(* Schneider Machine Expert - Basic project Shute_project, file version 2.2.0.0 *)
(* ProjectInformations: Name=Yeni proje *)

HARDWARE
  Cpu 0: TM221CE40R
  EthernetConfiguration: NetworkName=M221, IpAllocationMode=FixedAddress, IpAddress=0.0.0.0, SubnetMask=0.0.0.0
  SerialLineConfiguration: Baud=Baud19200, Parity=ParityEven, DataBits=DataBits8, StopBits=StopBits1, PhysicalMedium=PhysicalMediumRs485, TransmissionMode=TransmissionModeModbusRtu, SlaveId=1, Addressing=SlaveAddressing
  MastTask: UsePeriodScanMode=false, PeriodScan=100
  FastTask: Period=255
  CpuBehavior: StartingMode=StartAsPreviousState, AutoSaveRamOnEeprom=true, WatchdogPeriod=250

SYMBOLS  (address, symbol, comment, settings)
  %M0       K01_PERMISON
  %M1       K02_1_LOADING_ON
  %M2       K03_1_LEVEL_INDICATOR
  %M3       K04_1_TIMER
  %M4       K05_1_PARK_POSITION
  %M5       K06_1
  %M6       K07_1_SLACK_ROPE
  %M7       K08_1_LIFT_AUTO
  %M8       K11__1_LIFT_CHUTE
  %M9       K012_GAT1_O
  %M10      MAIN_CONTACTOR_1
  %M11      K017_1
  %M12      K12_1_OPEN_GATE
  %M13      K22_1_CLOSE_GATE
  %M14      K022_GATE_1_C
  %M15      LıFT_CHUTE_S63
  %M16      LOWER_CHUTE_S64
  %M17      LıFT_CHUTE_1
  %M18      LOADNG_ON
  %M19      K016_1_TIMER
  %M20      MAIN_CONTACTOR_2
  %M21      K07_2_SLACK_ROPE
  %M22      K02_2
  %M23      K06_2
  %M24      K05_2
  %M25      H62_LAMP
  %M26      ZS07_2
  %M27      K08_2
  %M28      K03_2
  %M29      K04_2
  %M30      LS01_2_SONDA_MAX_INPUT
  %M31      K012_2
  %M32      K022_2
  %M33      K016_2
  %M34      K017_2
  %I0.0     S61_EMERGENCY_OFF
  %I0.1     S62_EQUIPMENT_ON
  %I0.2     K100_K101_RELASE
  %I0.3     SLACK_ROPE_SENSOR_1
  %I0.4     LOADING_ON
  %I0.5     LOADING_OFF
  %I0.6     LIFT_CHUTE
  %I0.7     LOWER_CHUTE
  %I0.8     S65_LOADING_ON
  %I0.9     S66_LOADING_OFF
  %I0.10    ZS03_LIMIT_SWITCH_HOIST
  %I0.11    ZS07_LIMIT_PARK_SENSOR
  %I0.12    LS01_1_SONDA
  %I0.13    ZS01_1_LIMIT_SWITH_LOWER  "this should be 2zs01"
  %I0.14    GATE_1_1B11_O
  %I0.15    GATE_1_1B12
  %I0.16    GATE_2_2B11_O
  %I0.17    GATE_2_2B12_C
  %I0.18    S70_CHUTE_1
  %I0.19    S70_CHUTE_2
  %I0.20    ZS02_1
  %I0.21    SLACK_ROPE_SENSOR_2
  %I0.22    ZS02_2
  %I0.23    ZS072
  %Q0.0     H4_LAMP
  %Q0.1     H5_LAMP
  %Q0.2     H63_LAMP
  %Q0.3     K11_1_LIFT_CHUTE
  %Q0.4     K21_1_LOWER_CHUTE
  %Q0.5     K02_1_OUTPUT
  %Q0.6     K12_OPEN_GATE_1
  %Q0.7     K22_CLOSE_GATE_1
  %Q0.8     K11_2_LIFT_CHUTE
  %Q0.9     K12_2_LOWER_CHUTE
  %Q0.10    K02_2_OUTPUT
  %Q0.11    K12_OPEN_GATE_2
  %Q0.12    K22_2_CLOSE_GATE_2
  %Q0.13    K21_2

POU Yeni POU
  (* SectionNumber=1 *)

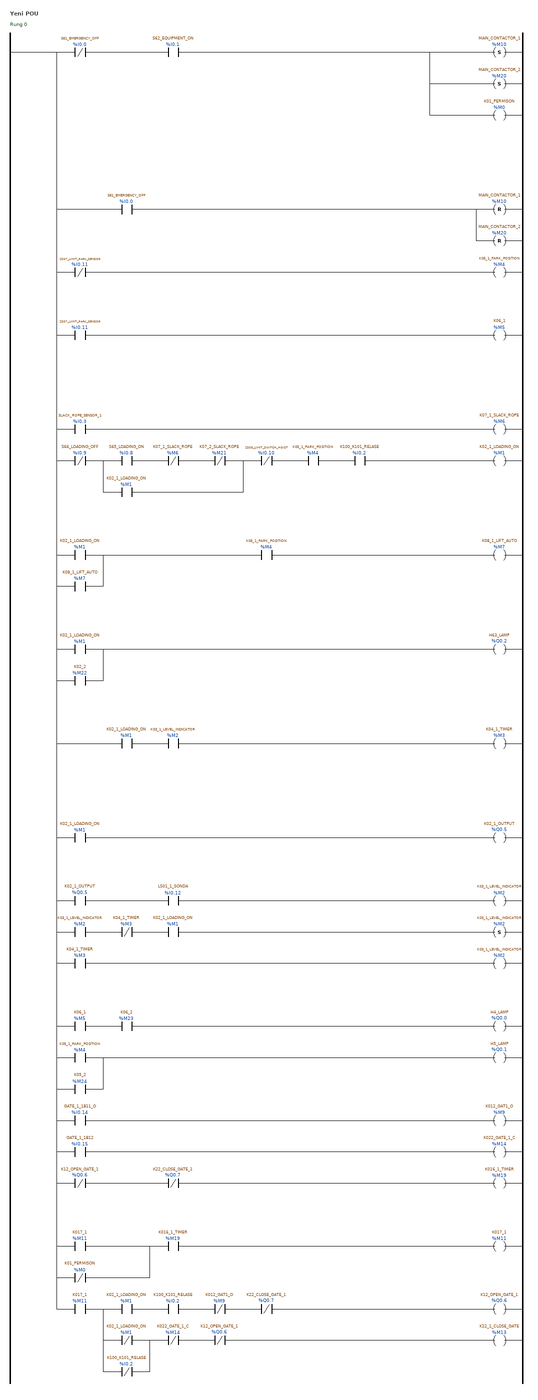

// Rung 0
  LD 1
  MPS
  ANDN %I0.0              (* S61_EMERGENCY_OFF *)
  AND %I0.1               (* S62_EQUIPMENT_ON *)
  S %M10                  (* MAIN_CONTACTOR_1 *)
  S %M20                  (* MAIN_CONTACTOR_2 *)
  ST %M0                  (* K01_PERMISON *)
  MRD
  AND %I0.0               (* S61_EMERGENCY_OFF *)
  R %M10                  (* MAIN_CONTACTOR_1 *)
  R %M20                  (* MAIN_CONTACTOR_2 *)
  MRD
  ANDN %I0.11             (* ZS07_LIMIT_PARK_SENSOR *)
  ST %M4                  (* K05_1_PARK_POSITION *)
  MRD
  AND %I0.11              (* ZS07_LIMIT_PARK_SENSOR *)
  ST %M5                  (* K06_1 *)
  MRD
  AND %I0.3               (* SLACK_ROPE_SENSOR_1 *)
  ST %M6                  (* K07_1_SLACK_ROPE *)
  MRD
  ANDN %I0.9              (* S66_LOADING_OFF *)
  AND( %I0.8              (* S65_LOADING_ON *)
  ANDN %M6                (* K07_1_SLACK_ROPE *)
  ANDN %M21               (* K07_2_SLACK_ROPE *)
  OR %M1                  (* K02_1_LOADING_ON *)
  )
  ANDN %I0.10             (* ZS03_LIMIT_SWITCH_HOIST *)
  AND %M4                 (* K05_1_PARK_POSITION *)
  AND %I0.2               (* K100_K101_RELASE *)
  ST %M1                  (* K02_1_LOADING_ON *)
  MRD
  AND( %M1                (* K02_1_LOADING_ON *)
  OR %M7                  (* K08_1_LIFT_AUTO *)
  )
  AND %M4                 (* K05_1_PARK_POSITION *)
  ST %M7                  (* K08_1_LIFT_AUTO *)
  MRD
  AND( %M1                (* K02_1_LOADING_ON *)
  OR %M22                 (* K02_2 *)
  )
  ST %Q0.2                (* H63_LAMP *)
  MRD
  AND %M1                 (* K02_1_LOADING_ON *)
  AND %M2                 (* K03_1_LEVEL_INDICATOR *)
  ST %M3                  (* K04_1_TIMER *)
  MRD
  AND %M1                 (* K02_1_LOADING_ON *)
  ST %Q0.5                (* K02_1_OUTPUT *)
  MRD
  AND %Q0.5               (* K02_1_OUTPUT *)
  AND %I0.12              (* LS01_1_SONDA *)
  ST %M2                  (* K03_1_LEVEL_INDICATOR *)
  MRD
  AND %M2                 (* K03_1_LEVEL_INDICATOR *)
  ANDN %M3                (* K04_1_TIMER *)
  AND %M1                 (* K02_1_LOADING_ON *)
  S %M2                   (* K03_1_LEVEL_INDICATOR *)
  MRD
  AND %M3                 (* K04_1_TIMER *)
  ST %M2                  (* K03_1_LEVEL_INDICATOR *)
  MRD
  AND %M5                 (* K06_1 *)
  AND %M23                (* K06_2 *)
  ST %Q0.0                (* H4_LAMP *)
  MRD
  AND( %M4                (* K05_1_PARK_POSITION *)
  OR %M24                 (* K05_2 *)
  )
  ST %Q0.1                (* H5_LAMP *)
  MRD
  AND %I0.14              (* GATE_1_1B11_O *)
  ST %M9                  (* K012_GAT1_O *)
  MRD
  AND %I0.15              (* GATE_1_1B12 *)
  ST %M14                 (* K022_GATE_1_C *)
  MRD
  ANDN %Q0.6              (* K12_OPEN_GATE_1 *)
  ANDN %Q0.7              (* K22_CLOSE_GATE_1 *)
  ST %M19                 (* K016_1_TIMER *)
  MRD
  AND( %M11               (* K017_1 *)
  ORN %M0                 (* K01_PERMISON *)
  )
  AND %M19                (* K016_1_TIMER *)
  ST %M11                 (* K017_1 *)
  MPP
  AND %M11                (* K017_1 *)
  MPS
  AND %M1                 (* K02_1_LOADING_ON *)
  AND %I0.2               (* K100_K101_RELASE *)
  ANDN %M9                (* K012_GAT1_O *)
  ANDN %Q0.7              (* K22_CLOSE_GATE_1 *)
  ST %Q0.6                (* K12_OPEN_GATE_1 *)
  MPP
  AND(N %M1               (* K02_1_LOADING_ON *)
  ORN %I0.2               (* K100_K101_RELASE *)
  )
  ANDN %M14               (* K022_GATE_1_C *)
  ANDN %Q0.6              (* K12_OPEN_GATE_1 *)
  ST %M13                 (* K22_1_CLOSE_GATE *)
  // as ST:
  //   IF NOT S61_EMERGENCY_OFF AND S62_EQUIPMENT_ON THEN MAIN_CONTACTOR_1 := TRUE; END_IF;
  //   IF NOT S61_EMERGENCY_OFF AND S62_EQUIPMENT_ON THEN MAIN_CONTACTOR_2 := TRUE; END_IF;
  //   K01_PERMISON := NOT S61_EMERGENCY_OFF AND S62_EQUIPMENT_ON;
  //   IF S61_EMERGENCY_OFF THEN MAIN_CONTACTOR_1 := FALSE; END_IF;
  //   IF S61_EMERGENCY_OFF THEN MAIN_CONTACTOR_2 := FALSE; END_IF;
  //   K05_1_PARK_POSITION := NOT ZS07_LIMIT_PARK_SENSOR;
  //   K06_1 := ZS07_LIMIT_PARK_SENSOR;
  //   K07_1_SLACK_ROPE := SLACK_ROPE_SENSOR_1;
  //   K02_1_LOADING_ON := NOT S66_LOADING_OFF AND (S65_LOADING_ON AND NOT K07_1_SLACK_ROPE AND NOT K07_2_SLACK_ROPE OR K02_1_LOADING_ON) AND NOT ZS03_LIMIT_SWITCH_HOIST AND K05_1_PARK_POSITION AND K100_K101_RELASE;
  //   K08_1_LIFT_AUTO := (K02_1_LOADING_ON OR K08_1_LIFT_AUTO) AND K05_1_PARK_POSITION;
  //   H63_LAMP := K02_1_LOADING_ON OR K02_2;
  //   K04_1_TIMER := K02_1_LOADING_ON AND K03_1_LEVEL_INDICATOR;
  //   K02_1_OUTPUT := K02_1_LOADING_ON;
  //   K03_1_LEVEL_INDICATOR := K02_1_OUTPUT AND LS01_1_SONDA;
  //   IF K03_1_LEVEL_INDICATOR AND NOT K04_1_TIMER AND K02_1_LOADING_ON THEN K03_1_LEVEL_INDICATOR := TRUE; END_IF;
  //   K03_1_LEVEL_INDICATOR := K04_1_TIMER;
  //   H4_LAMP := K06_1 AND K06_2;
  //   H5_LAMP := K05_1_PARK_POSITION OR K05_2;
  //   K012_GAT1_O := GATE_1_1B11_O;
  //   K022_GATE_1_C := GATE_1_1B12;
  //   K016_1_TIMER := NOT K12_OPEN_GATE_1 AND NOT K22_CLOSE_GATE_1;
  //   K017_1 := (K017_1 OR NOT K01_PERMISON) AND K016_1_TIMER;
  //   K12_OPEN_GATE_1 := K017_1 AND K02_1_LOADING_ON AND K100_K101_RELASE AND NOT K012_GAT1_O AND NOT K22_CLOSE_GATE_1;
  //   K22_1_CLOSE_GATE := K017_1 AND (NOT K02_1_LOADING_ON OR NOT K100_K101_RELASE) AND NOT K022_GATE_1_C AND NOT K12_OPEN_GATE_1;

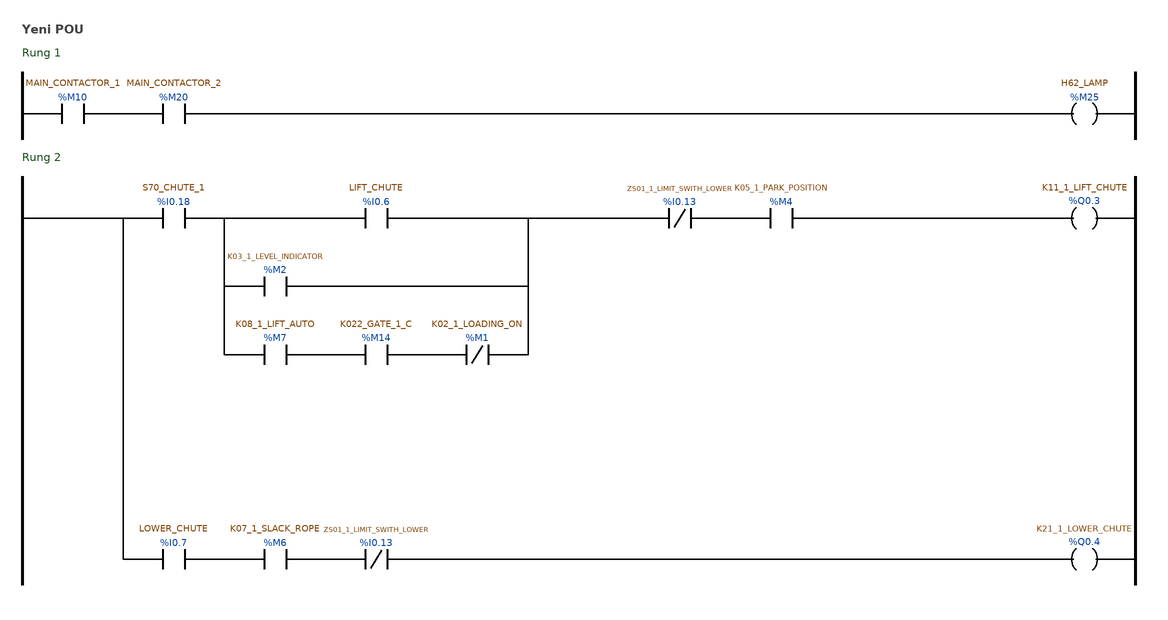

// Rung 1
  LD %M10                 (* MAIN_CONTACTOR_1 *)
  AND %M20                (* MAIN_CONTACTOR_2 *)
  ST %M25                 (* H62_LAMP *)
  // as ST:
  //   H62_LAMP := MAIN_CONTACTOR_1 AND MAIN_CONTACTOR_2;

// Rung 2
  LD 1
  MPS
  AND %I0.18              (* S70_CHUTE_1 *)
  AND( %I0.6              (* LIFT_CHUTE *)
  OR( %M2                 (* K03_1_LEVEL_INDICATOR *)
  OR( %M7                 (* K08_1_LIFT_AUTO *)
  AND %M14                (* K022_GATE_1_C *)
  ANDN %M1                (* K02_1_LOADING_ON *)
  )
  )
  )
  ANDN %I0.13             (* ZS01_1_LIMIT_SWITH_LOWER *)
  AND %M4                 (* K05_1_PARK_POSITION *)
  ST %Q0.3                (* K11_1_LIFT_CHUTE *)
  MPP
  AND %I0.7               (* LOWER_CHUTE *)
  AND %M6                 (* K07_1_SLACK_ROPE *)
  ANDN %I0.13             (* ZS01_1_LIMIT_SWITH_LOWER *)
  ST %Q0.4                (* K21_1_LOWER_CHUTE *)
  // as ST:
  //   K11_1_LIFT_CHUTE := S70_CHUTE_1 AND (LIFT_CHUTE OR K03_1_LEVEL_INDICATOR OR K08_1_LIFT_AUTO AND K022_GATE_1_C AND NOT K02_1_LOADING_ON) AND NOT ZS01_1_LIMIT_SWITH_LOWER AND K05_1_PARK_POSITION;
  //   K21_1_LOWER_CHUTE := LOWER_CHUTE AND K07_1_SLACK_ROPE AND NOT ZS01_1_LIMIT_SWITH_LOWER;

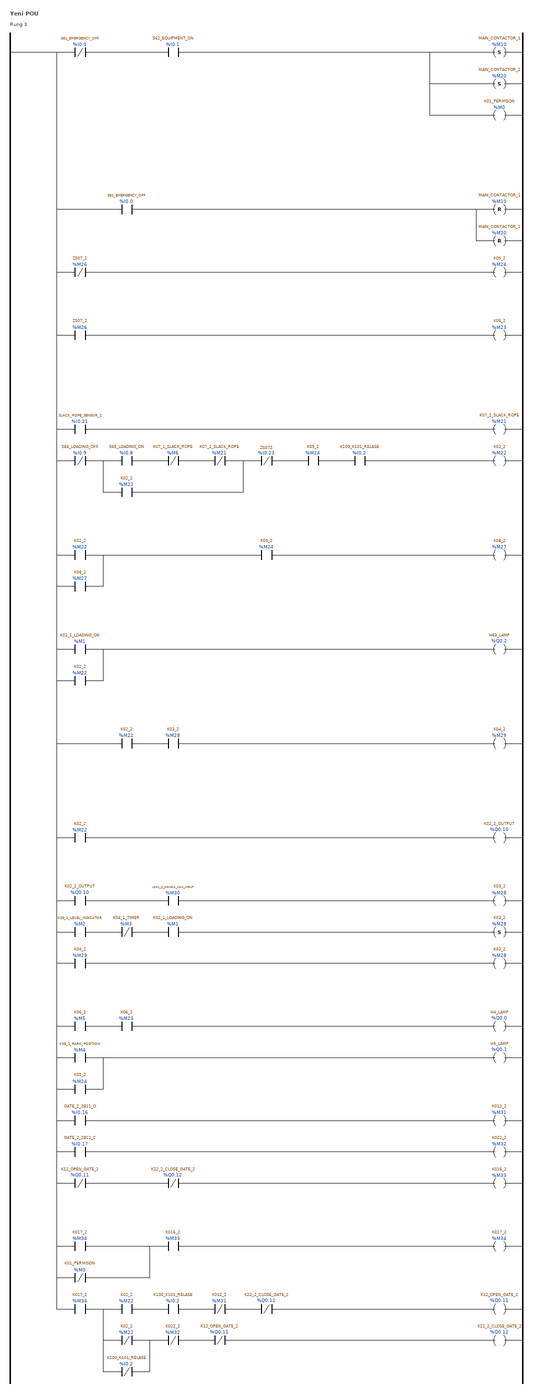

// Rung 3
  LD 1
  MPS
  ANDN %I0.0              (* S61_EMERGENCY_OFF *)
  AND %I0.1               (* S62_EQUIPMENT_ON *)
  S %M10                  (* MAIN_CONTACTOR_1 *)
  S %M20                  (* MAIN_CONTACTOR_2 *)
  ST %M0                  (* K01_PERMISON *)
  MRD
  AND %I0.0               (* S61_EMERGENCY_OFF *)
  R %M10                  (* MAIN_CONTACTOR_1 *)
  R %M20                  (* MAIN_CONTACTOR_2 *)
  MRD
  ANDN %M26               (* ZS07_2 *)
  ST %M24                 (* K05_2 *)
  MRD
  AND %M26                (* ZS07_2 *)
  ST %M23                 (* K06_2 *)
  MRD
  AND %I0.21              (* SLACK_ROPE_SENSOR_2 *)
  ST %M21                 (* K07_2_SLACK_ROPE *)
  MRD
  ANDN %I0.9              (* S66_LOADING_OFF *)
  AND( %I0.8              (* S65_LOADING_ON *)
  ANDN %M6                (* K07_1_SLACK_ROPE *)
  ANDN %M21               (* K07_2_SLACK_ROPE *)
  OR %M22                 (* K02_2 *)
  )
  ANDN %I0.23             (* ZS072 *)
  AND %M24                (* K05_2 *)
  AND %I0.2               (* K100_K101_RELASE *)
  ST %M22                 (* K02_2 *)
  MRD
  AND( %M22               (* K02_2 *)
  OR %M27                 (* K08_2 *)
  )
  AND %M24                (* K05_2 *)
  ST %M27                 (* K08_2 *)
  MRD
  AND( %M1                (* K02_1_LOADING_ON *)
  OR %M22                 (* K02_2 *)
  )
  ST %Q0.2                (* H63_LAMP *)
  MRD
  AND %M22                (* K02_2 *)
  AND %M28                (* K03_2 *)
  ST %M29                 (* K04_2 *)
  MRD
  AND %M22                (* K02_2 *)
  ST %Q0.10               (* K02_2_OUTPUT *)
  MRD
  AND %Q0.10              (* K02_2_OUTPUT *)
  AND %M30                (* LS01_2_SONDA_MAX_INPUT *)
  ST %M28                 (* K03_2 *)
  MRD
  AND %M2                 (* K03_1_LEVEL_INDICATOR *)
  ANDN %M3                (* K04_1_TIMER *)
  AND %M1                 (* K02_1_LOADING_ON *)
  S %M28                  (* K03_2 *)
  MRD
  AND %M29                (* K04_2 *)
  ST %M28                 (* K03_2 *)
  MRD
  AND %M5                 (* K06_1 *)
  AND %M23                (* K06_2 *)
  ST %Q0.0                (* H4_LAMP *)
  MRD
  AND( %M4                (* K05_1_PARK_POSITION *)
  OR %M24                 (* K05_2 *)
  )
  ST %Q0.1                (* H5_LAMP *)
  MRD
  AND %I0.16              (* GATE_2_2B11_O *)
  ST %M31                 (* K012_2 *)
  MRD
  AND %I0.17              (* GATE_2_2B12_C *)
  ST %M32                 (* K022_2 *)
  MRD
  ANDN %Q0.11             (* K12_OPEN_GATE_2 *)
  ANDN %Q0.12             (* K22_2_CLOSE_GATE_2 *)
  ST %M33                 (* K016_2 *)
  MRD
  AND( %M34               (* K017_2 *)
  ORN %M0                 (* K01_PERMISON *)
  )
  AND %M33                (* K016_2 *)
  ST %M34                 (* K017_2 *)
  MPP
  AND %M34                (* K017_2 *)
  MPS
  AND %M22                (* K02_2 *)
  AND %I0.2               (* K100_K101_RELASE *)
  ANDN %M31               (* K012_2 *)
  ANDN %Q0.12             (* K22_2_CLOSE_GATE_2 *)
  ST %Q0.11               (* K12_OPEN_GATE_2 *)
  MPP
  AND(N %M22              (* K02_2 *)
  ORN %I0.2               (* K100_K101_RELASE *)
  )
  ANDN %M32               (* K022_2 *)
  ANDN %Q0.11             (* K12_OPEN_GATE_2 *)
  ST %Q0.12               (* K22_2_CLOSE_GATE_2 *)
  // as ST:
  //   IF NOT S61_EMERGENCY_OFF AND S62_EQUIPMENT_ON THEN MAIN_CONTACTOR_1 := TRUE; END_IF;
  //   IF NOT S61_EMERGENCY_OFF AND S62_EQUIPMENT_ON THEN MAIN_CONTACTOR_2 := TRUE; END_IF;
  //   K01_PERMISON := NOT S61_EMERGENCY_OFF AND S62_EQUIPMENT_ON;
  //   IF S61_EMERGENCY_OFF THEN MAIN_CONTACTOR_1 := FALSE; END_IF;
  //   IF S61_EMERGENCY_OFF THEN MAIN_CONTACTOR_2 := FALSE; END_IF;
  //   K05_2 := NOT ZS07_2;
  //   K06_2 := ZS07_2;
  //   K07_2_SLACK_ROPE := SLACK_ROPE_SENSOR_2;
  //   K02_2 := NOT S66_LOADING_OFF AND (S65_LOADING_ON AND NOT K07_1_SLACK_ROPE AND NOT K07_2_SLACK_ROPE OR K02_2) AND NOT ZS072 AND K05_2 AND K100_K101_RELASE;
  //   K08_2 := (K02_2 OR K08_2) AND K05_2;
  //   H63_LAMP := K02_1_LOADING_ON OR K02_2;
  //   K04_2 := K02_2 AND K03_2;
  //   K02_2_OUTPUT := K02_2;
  //   K03_2 := K02_2_OUTPUT AND LS01_2_SONDA_MAX_INPUT;
  //   IF K03_1_LEVEL_INDICATOR AND NOT K04_1_TIMER AND K02_1_LOADING_ON THEN K03_2 := TRUE; END_IF;
  //   K03_2 := K04_2;
  //   H4_LAMP := K06_1 AND K06_2;
  //   H5_LAMP := K05_1_PARK_POSITION OR K05_2;
  //   K012_2 := GATE_2_2B11_O;
  //   K022_2 := GATE_2_2B12_C;
  //   K016_2 := NOT K12_OPEN_GATE_2 AND NOT K22_2_CLOSE_GATE_2;
  //   K017_2 := (K017_2 OR NOT K01_PERMISON) AND K016_2;
  //   K12_OPEN_GATE_2 := K017_2 AND K02_2 AND K100_K101_RELASE AND NOT K012_2 AND NOT K22_2_CLOSE_GATE_2;
  //   K22_2_CLOSE_GATE_2 := K017_2 AND (NOT K02_2 OR NOT K100_K101_RELASE) AND NOT K022_2 AND NOT K12_OPEN_GATE_2;

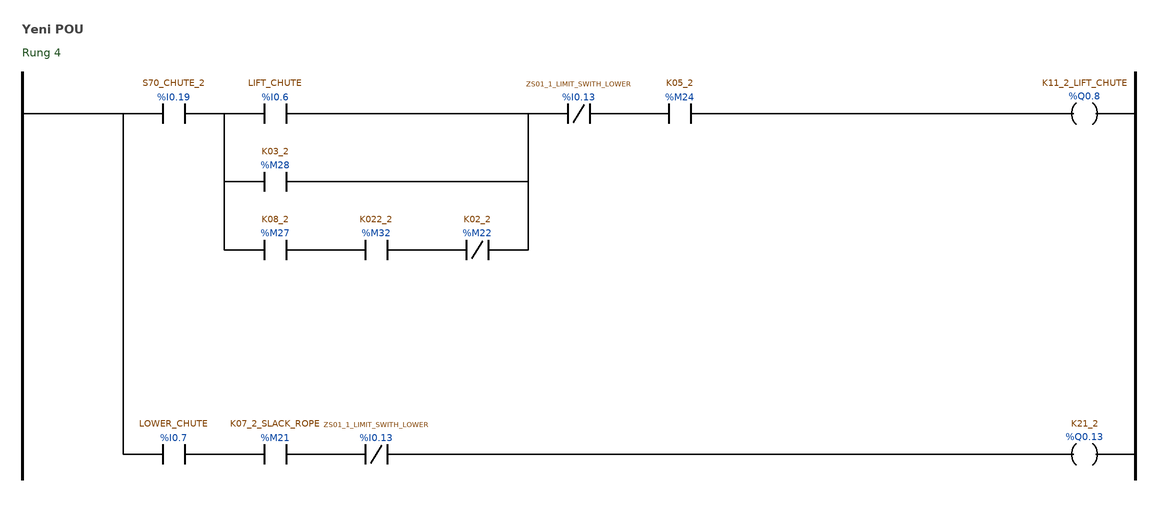

// Rung 4
  LD 1
  MPS
  AND %I0.19              (* S70_CHUTE_2 *)
  AND( %I0.6              (* LIFT_CHUTE *)
  OR( %M28                (* K03_2 *)
  OR( %M27                (* K08_2 *)
  AND %M32                (* K022_2 *)
  ANDN %M22               (* K02_2 *)
  )
  )
  )
  ANDN %I0.13             (* ZS01_1_LIMIT_SWITH_LOWER *)
  AND %M24                (* K05_2 *)
  ST %Q0.8                (* K11_2_LIFT_CHUTE *)
  MPP
  AND %I0.7               (* LOWER_CHUTE *)
  AND %M21                (* K07_2_SLACK_ROPE *)
  ANDN %I0.13             (* ZS01_1_LIMIT_SWITH_LOWER *)
  ST %Q0.13               (* K21_2 *)
  // as ST:
  //   K11_2_LIFT_CHUTE := S70_CHUTE_2 AND (LIFT_CHUTE OR K03_2 OR K08_2 AND K022_2 AND NOT K02_2) AND NOT ZS01_1_LIMIT_SWITH_LOWER AND K05_2;
  //   K21_2 := LOWER_CHUTE AND K07_2_SLACK_ROPE AND NOT ZS01_1_LIMIT_SWITH_LOWER;
